// TIA Portal V19 export
FUNCTION "FC_IncHub" : Void   // FC208, STL
TITLE = Absolut-Wegmessung Hub
{ S7_Optimized_Access := 'FALSE' }
// stored: AutoNumber false
   VAR_INPUT
      Eingangswert : DInt;   // kompletter Eingangswert
      Direction : Byte;
      Offset : DInt;
      Anz_FM : Int;   // Anzahl Fehlmessungen
      Faktor_Umrechnung : Real;   // Umrechnung in mm
   END_VAR
   VAR_IN_OUT
      Alarm : Bool;
      count : Byte;
      Messwert : DInt;   // Messwert in mm
   END_VAR
   VAR_TEMP
      Messung : DInt;   // neuer gemessener Wert
      invers : Bool;
   END_VAR
BEGIN

NETWORK
TITLE = 
//-----------------
//    Messwert
//-----------------
      L     0;
      L     #Direction;
      <>I;
      =     #invers;

      L     #Eingangswert;
      T     #Messung;
      L     0;
      <>D;
      JC    ok;

      L     #Anz_FM;
      L     #count;
      <=I;
      JC    err;
      +     1;
      T     #count;
      BE;
err:  SET;
      S     #Alarm;
      BE;

ok:   SET;
      R     #Alarm;

      L     0;
      T     #count;

      L     #Messung;
      AN    #invers;
      JC    sub;
      INVD;
sub:  DTR;
      L     #Faktor_Umrechnung;
      *R;
      RND;
      L     #Offset;
      +D;
      T     #Messwert;
      BE;

END_FUNCTION
